TYPE Array8_LReal :
UNION
	arrByte			:ARRAY[0..7] OF BYTE;
	rValue			:LREAL;
END_UNION
END_TYPE

(* stored: Version 1.1.0.1
   DUT Array8_LReal: Id {ed274fc9-6308-4891-b7cf-a95f32782fb7} *)
